TYPE ST_TempLoad_State :
STRUCT
	bPparamLoaded: BOOL;
	bMparamLoaded: BOOL;
	bPparamLoad: BOOL;
	bMparamLoad: BOOL;
	bSupplyParamsLoad: BOOL;
	bSupplyParamsLoaded: BOOL;
END_STRUCT
END_TYPE

(* stored: Version 1.1.0.1, ProductVersion 3.1.0.26
   DUT ST_TempLoad_State: Id {b8061634-8fd3-4a37-acd0-98f326ca15a3} *)
